PROGRAM MAIN
VAR
END_VAR

END_PROGRAM

(* stored: Version 1.1.0.1, ProductVersion 3.1.0.36
   POU MAIN: Id {a2663345-514a-4133-b25f-40109ea5277d} *)
